RoboDK station: EjercicioRobot4.rdk

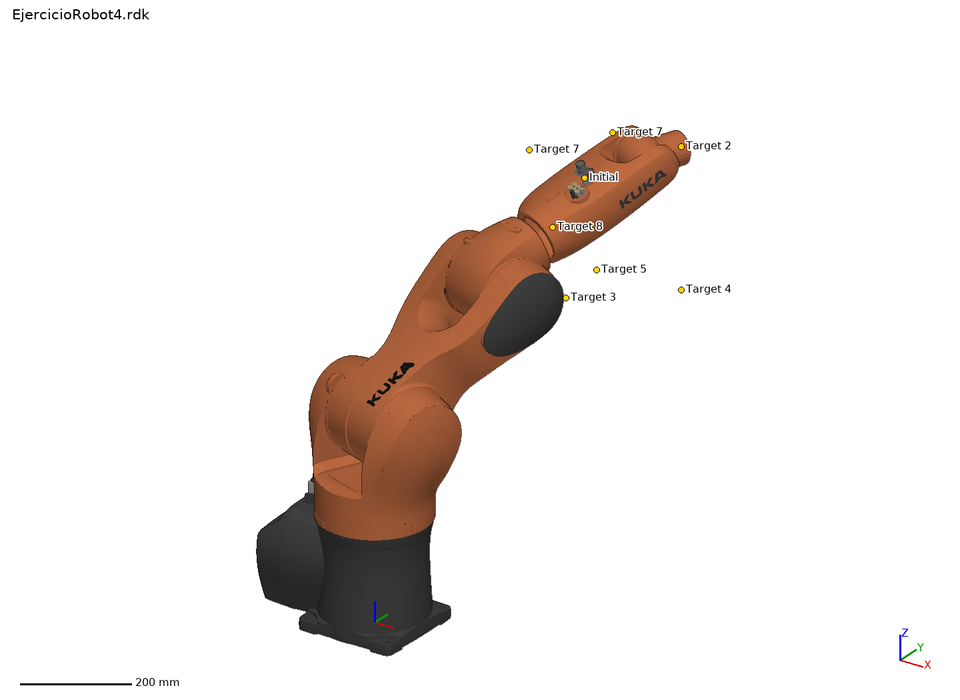
[picture v0: the station drawn from its stored meshes, robots at their saved joint values, targets as dots, program paths as lines]
Station EjercicioRobot4 (saved by RoboDK 6.0.4). Poses are relative to the parent item; angles as X-Y-Z fixed-axis rotations.
  - frame KUKA KR 6 R700 sixx Base at (0, 0, 0) mm
    - robot KUKA KR 6 R700 sixx: 6 axes, payload 6 kg, reach 706.7 mm, repeatability 0.03 mm, weight 50 kg
        modified DH rows (alpha deg, a mm, theta deg, d mm): 0, 0, 0, 400; -90, 25, 0, 0; 0, 315, -90, 0; -90, 35, 0, 365; 90, 0, 0, 0; -90, 0, 180, 80
        joint limits [-170, -190, -120, -185, -120, -350] to [170, 45, 156, 185, 120, 350]; home [0, -90, 90, 0, 0, 0]; saved at [-71.64, -37.979, 18.25, 0, 19.729, 0]
    - target Initial (Cartesian target) at (148.06, 446.13, 750) mm, rotated rx 0 ry 90 rz 71.64 deg; joints [-71.64, -89.99, 89.99, 0, 0, 0] of KUKA KR 6 R700 sixx
    - target Target 2 (Cartesian target) at (215.78, 650.18, 750) mm, rotated rx 0 ry 90 rz 71.64 deg; joints [-71.64, -37.979, 18.25, 0, 19.729, 0] of KUKA KR 6 R700 sixx
    - target Target 3 (Cartesian target) at (134.79, 406.15, 522.81) mm, rotated rx -180 ry 60 rz -108.36 deg; joints [-71.64, -89.99, 119.99, 0, 0, 0] of KUKA KR 6 R700 sixx
    - target Target 4 (Cartesian target) at (222.96, 640.87, 470.19) mm, rotated rx -98.77 ry -12.36 rz -16.47 deg; joints [-70.709, -42.573, 68.981, 3.003, -17.86, 99.78] of KUKA KR 6 R700 sixx
    - target Target 5 (Cartesian target) at (-11.23, 710.1, 416.69) mm, rotated rx -98.77 ry -12.36 rz -16.47 deg; joints [-93.258, -31.089, 58.01, -52.126, -27.485, 147.879] of KUKA KR 6 R700 sixx
    - target Target 7 (Cartesian target) at (15.61, 721.06, 693.66) mm, rotated rx -77.59 ry -4.09 rz -19.55 deg; joints [-90.83, -27.147, 11.393, 82.357, 19.183, 16.614] of KUKA KR 6 R700 sixx
    - target Target 7 (Cartesian target) at (-18, 509.79, 734.17) mm, rotated rx -69.67 ry 0.03 rz -21.66 deg; joints [-95.93, -80.72, 86.9, -44.98, -37.93, 138.51] of KUKA KR 6 R700 sixx
    - target Target 8 (Cartesian target) at (-26.95, 595.84, 543.03) mm, rotated rx -88.06 ry -9.33 rz -20.15 deg; joints [-95.93, -60.17, 86.9, -44.98, -37.92, 138.51] of KUKA KR 6 R700 sixx
  - Python program Prog1 (listed below)

--- Python program Prog1 ---
# Type help("robodk.robolink") or help("robodk.robomath") for more information
# Press F5 to run the script
# Documentation: https://robodk.com/doc/en/RoboDK-API.html
# Reference:     https://robodk.com/doc/en/PythonAPI/robodk.html
# Note: It is not required to keep a copy of this file, your Python script is saved with your RDK project

# You can also use the new version of the API:
from robodk import robolink    # RoboDK API
from robodk import robomath    # Robot toolbox
RDK = robolink.Robolink()

# Forward and backwards compatible use of the RoboDK API:
# Remove these 2 lines to follow python programming guidelines
from robodk import *      # RoboDK API
from robolink import *    # Robot toolbox
# Link to RoboDK
# RDK = Robolink()

# Notify user:
print('To edit this program:\nright click on the Python program, then, select "Edit Python script"')

# Program example:
item = RDK.Item('base')
if item.Valid():
    print('Item selected: ' + item.Name())
    print('Item posistion: ' + repr(item.Pose()))

print('Items in the station:')
itemlist = RDK.ItemList()
print(itemlist)

# Provoking an exception will display the console output if you run this script from RoboDK
raise Exception('Program not edited.')
